SUBAPPLICATION Softkey2_TO_A2X2_BG (* 2 VT-SoftKeys (Softkey_IXA, Hoch/Runter) gebuendelt auf einen einzigen bidirektionalen A2X2-Adapterausgang: Tastendruecke gehen ueber A2X2_4AX_TO_2X nach draussen, der ueber denselben Adapter zurueckkommende, tatsaechlich erreichte Zustand faerbt beide SoftKeys per GreenWhiteBackground1_AX - 'SUB style': das Buendeln steckt im Composite, nicht in der Resource des Geraets. *)
  (* Standard: 61499-2; Description: Copyright (c) 2026 HR Agrartechnik GmbH This program and the accompanying materials are made available under the terms of the Eclipse Public License 2.0 which is available at https://www.eclipse.org/legal/epl-2.0/ SPDX-License-Identifier: EPL-2.0 *)
  (* Version 1.0, 2026-09-05, Franz Höpfinger, HR Agrartechnik GmbH, initial API and implementation and/or initial documentation *)
  PACKAGE MyLib::sys;
  IMPORT isobus::UT::Q::const::IDs::ID_NULL;
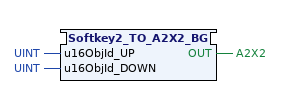
  VAR_INPUT
    u16ObjId_UP : UINT := ID_NULL; (* Object ID SoftKey Hoch (traegt auch das GreenWhiteBackground) *)
    u16ObjId_DOWN : UINT := ID_NULL; (* Object ID SoftKey Runter (traegt auch das GreenWhiteBackground) *)
  END_VAR
  PLUGS
    OUT : adapter::types::bidirectional::A2X2; (* Gebuendelter Roundtrip: sendet UP/DOWN-Tastendruecke, empfaengt UP/DOWN-Rueckmeldezustand *)
  END_PLUGS
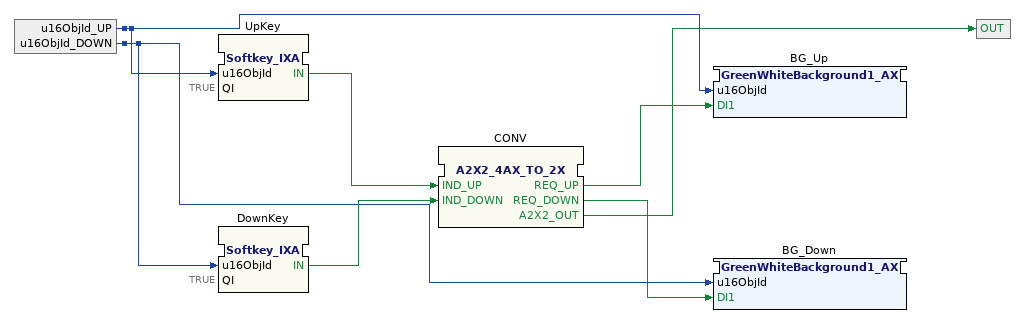
  FBS
    UpKey : isobus::UT::io::Softkey::Softkey_IXA(QI := TRUE);
    DownKey : isobus::UT::io::Softkey::Softkey_IXA(QI := TRUE);
    CONV : adapter::conversion::bidirectional::A2X2_4AX_TO_2X;
  END_FBS
  SUBAPPS
    BG_Up : MyLib::sys::GreenWhiteBackground1_AX;
    BG_Down : MyLib::sys::GreenWhiteBackground1_AX;
  END_SUBAPPS
  DATA_CONNECTIONS
    u16ObjId_UP TO UpKey.u16ObjId;
    u16ObjId_DOWN TO DownKey.u16ObjId;
    u16ObjId_UP TO BG_Up.u16ObjId;
    u16ObjId_DOWN TO BG_Down.u16ObjId;
  END_CONNECTIONS
  ADAPTER_CONNECTIONS
    UpKey.IN TO CONV.IND_UP;
    DownKey.IN TO CONV.IND_DOWN;
    CONV.REQ_UP TO BG_Up.DI1;
    CONV.REQ_DOWN TO BG_Down.DI1;
    CONV.A2X2_OUT TO OUT;
  END_CONNECTIONS
END_SUBAPPLICATION
